{attribute addProperty BoxType "EL3101-0000-0018"}
{attribute addProperty Id "StatusAT %I*Status_845218981621ValueAT %I*INT16217"}
{attribute addProperty CRC "142569927"}
{attribute addProperty SizeInBites "32"}
{attribute addProperty SizeInBytes "4"}
TYPE AI_Standard_087F71C7 :
STRUCT
	{attribute addProperty Name "Status"}
	Status AT %I* : Status_84521898;
	{attribute addProperty Name "Value"}
	Value AT %I* : INT;
END_STRUCT
END_TYPE

(* stored: Version 1.2.0.0, ProductVersion 3.1.4024.9
   DUT AI_Standard_087F71C7: Id {695019e0-a23e-4064-b050-44e97df5e44f} *)
